// TIA Portal V20 export
TYPE "UDT_Interlock_HAI"
   STRUCT
      PickUp_OK : Bool;
      Loading_Completion : Bool;
      "Byte0.bit2" : Bool;
      "Byte0.bit3" : Bool;
      "Byte0.bit4" : Bool;
      "Byte0.bit5" : Bool;
      "Byte0.bit6" : Bool;
      "Byte0.bit7" : Bool;
      Deposit_Ok : Bool;
      Unloading_Completion : Bool;
      Byte1_bit2 : Bool;
      Byte1_bit3 : Bool;
      Byte1_bit4 : Bool;
      Byte1_bit5 : Bool;
      Byte1_bit6 : Bool;
      Byte1_bit7 : Bool;
      Byte2_bit0 : Bool;
      Byte2_bit1 : Bool;
      Byte2_bit2 : Bool;
      Byte2_bit3 : Bool;
      Byte2_bit4 : Bool;
      Byte2_bit5 : Bool;
      Byte2_bit6 : Bool;
      Byte2_bit7 : Bool;
      Byte3_bit0 : Bool;
      Byte3_bit1 : Bool;
      Byte3_bit2 : Bool;
      Byte3_bit3 : Bool;
      Byte3_bit4 : Bool;
      Byte3_bit5 : Bool;
      Byte3_bit6 : Bool;
      Byte3_bit7 : Bool;
   END_STRUCT;
END_TYPE
